// TIA Portal project "programa_plc_hmi_V16" (V16)

(* hardware
DEVICE "S71500/ET200MP station_1"  S7-1500 station
   slot 0: "Rail_0"  Rack  6ES7 590-1***0-0AA0
   slot 1: "PLC_1"  CPU 1513-1 PN  6ES7 513-1AL02-0AB0  V2.6
      slot 3: "CPU display_1"  6ES7591-1AA00-0AA0
   slot 2: "DI 16x24VDC BA_1"  DI 16x24VDC BA  6ES7 521-1BH10-0AA0  V1.0
   slot 3: "DQ 16x24VDC/0.5A BA_1"  DQ 16x24VDC/0.5A BA  6ES7 522-1BH10-0AA0  V1.0
   slot 4: "AI 4xU/I/RTD/TC / AQ 2xU/I ST_1"  AI/AQ 4xU/I/RTD/TC / 2xU/I ST  6ES7 534-7QE00-0AB0  V1.0
DEVICE "HMI_1"  KTP400 Comfort
   slot 0: "HMI_1"  KTP400 Comfort  6AV2 124-2DC01-0AX0  16.0.0.0
   slot 1: "HMI_RT_1"  KTP400 Comfort  6AV2 124-2DC01-0AX0  16.0.0.0
   slot 5: "HMI_1.IE_CP_1"  PROFINET Interface  16.0.0.0
      slot 1: "Interfaz PROFINET_1"  PROFINET Interface
         slot 1: "Port_1"  Port
   slot 7: "HMI_1.MPI/DP_CP_1"  MPI/DP Interface  16.0.0.0
*)

// ===== PLC "PLC_1"  CPU 1513-1 PN =====

VAR_GLOBAL   // PLC tag table "Default tag table"
   "System_Byte" AT %MB1 : Byte;
   "FirstScan" AT %M1.0 : Bool;
   "DiagStatusUpdate" AT %M1.1 : Bool;
   "AlwaysTRUE" AT %M1.2 : Bool;
   "AlwaysFALSE" AT %M1.3 : Bool;
   "Clock_Byte" AT %MB0 : Byte;
   "Clock_10Hz" AT %M0.0 : Bool;
   "Clock_5Hz" AT %M0.1 : Bool;
   "Clock_2.5Hz" AT %M0.2 : Bool;
   "Clock_2Hz" AT %M0.3 : Bool;
   "Clock_1.25Hz" AT %M0.4 : Bool;
   "Clock_1Hz" AT %M0.5 : Bool;
   "Clock_0.625Hz" AT %M0.6 : Bool;
   "Clock_0.5Hz" AT %M0.7 : Bool;
   "hmi star" AT %M200.0 : Bool;
   "hm1 led" AT %M200.1 : Bool;
END_VAR

VAR_GLOBAL   // PLC tag table "Conveyor_1"
   "c1_paro_de_emergencia" AT %I0.0 : Bool;
   "c1_barrera_de_seguridad" AT %I0.1 : Bool;
   "c1_variador_en_run" AT %I0.2 : Bool;
   "c1_auxiliar_guardamotor" AT %I0.3 : Bool;
   "c1_auxiliar_seccionador" AT %I0.4 : Bool;
   "c1_variador_en_falla" AT %I0.5 : Bool;
   "c1_pulsador_arranque" AT %I0.6 : Bool;
   "c1_pulsador_parada" AT %I0.7 : Bool;
   "c1_reset" AT %I1.0 : Bool;
   "c1_modo_auto_manual" AT %I1.1 : Bool;
   "c1_variador_a_run" AT %Q0.0 : Bool;
   "c1_sistema_en_automatico" AT %Q0.1 : Bool;
   "c1_sistema_en_manual" AT %Q0.2 : Bool;
   "c1_sistema_en_falla" AT %Q0.3 : Bool;
   "c1_sirena" AT %Q0.4 : Bool;
   "c1_reset_sistema" AT %Q0.5 : Bool;
   "c1_referencia_de_velocidad" AT %IW2 : Int;
   "c1_referencia_actual_velocidad" AT %QW2 : Int;
   "c1_falla_en_arraque" AT %M110.0 : Bool;
   "c1_auxiliar_conveyor_run" AT %M110.1 : Bool;
   "c1_indicador_conveyor_run" AT %Q0.6 : Bool;
   "c1_auxiliar_modo_automatico" AT %M110.3 : Bool;
   "c1_auxiliar_modo_manual" AT %M110.4 : Bool;
   "c1_auxiliar_start_manual" AT %M110.5 : Bool;
   "c1_auxiliar_start_auto" AT %M110.6 : Bool;
   "c1_paro_de_emergencia_m" AT %M100.0 : Bool;
   "c1_barrera_de_seguridad_m" AT %M100.1 : Bool;
   "c1_variador_en_run_m" AT %M100.2 : Bool;
   "c1_auxiliar_guardamotor_m" AT %M100.3 : Bool;
   "c1_auxiliar_seccionador_m" AT %M100.4 : Bool;
   "c1_variador_en_falla_m" AT %M100.5 : Bool;
   "c1_pulsador_arranque_m" AT %M100.6 : Bool;
   "c1_pulsador_parada_m" AT %M100.7 : Bool;
   "c1_reset_m" AT %M101.0 : Bool;
   "c1_modo_auto_manual_m" AT %M101.1 : Bool;
   "c1_variador_a_run_m" AT %M105.0 : Bool;
   "c1_sistema_en_automatico_m" AT %M105.1 : Bool;
   "c1_sistema_en_manual_m" AT %M105.2 : Bool;
   "c1_sistema_en_falla_m" AT %M105.3 : Bool;
   "c1_sirena_m" AT %M105.4 : Bool;
   "c1_reset_sistema_m" AT %M105.5 : Bool;
   "c1_indicador_conveyor_run_m" AT %M105.6 : Bool;
   "c1_referencia_de_velocidad_m" AT %MW150 : Word;
   "c1_referencia_actual_velocidad_m" AT %MW170 : Word;
   "c1_percentage input" AT %MW160 : Word;
   "c1_brazo_en_funcionamiento" AT %I1.2 : Bool;
   "c1_brazo_en_falla" AT %I1.3 : Bool;
   "c1_cnc_funcionamiento" AT %I1.4 : Bool;
   "c1_brazo_en_funcionamiento_m" AT %M101.2 : Bool;
   "c1_brazo_en_falla_m" AT %M101.3 : Bool;
   "c1_cnc_funcionamiento_m" AT %M101.4 : Bool;
   "c1_selector_producto" AT %Q0.7 : Bool;
   "c1_selector_producto_m" AT %M105.7 : Bool;
   "c1_sistema_cnc_1_en _funcinamiento" AT %M110.7 : Bool;
   "c1_sistema_cnc_1_en_falla" AT %M111.0 : Bool;
   "c1_sensor_producto_acabado" AT %I1.5 : Bool;
   "c1_sensor_producto_acabado_m" AT %M101.5 : Bool;
   "c1_cnc_arranque" AT %Q1.0 : Bool;
   "c1_cnc_parada" AT %Q1.1 : Bool;
   "c1_cnc_reset" AT %Q1.2 : Bool;
   "c1_cnc_arranque_m" AT %M106.0 : Bool;
   "c1_cnc_parada_m" AT %M106.1 : Bool;
   "c1_cnc_reset_m" AT %M106.2 : Bool;
   "c1_sensor_producto_entrada" AT %I1.6 : Bool;
   "c1_sensor_producto_entrada_m" AT %M101.6 : Bool;
   "c1_habilitar_material" AT %Q1.3 : Bool;
   "c1_habilitar_material_m" AT %M106.3 : Bool;
   "c1hmistart" AT %M210.0 : Bool;
   "c1hmiled" AT %M210.1 : Bool;
END_VAR

DATA_BLOCK "Direct_start_conveyor_1"   // DB1
{ S7_Optimized_Access := 'TRUE' }
VERSION : 0.1
// stored: InstanceOfName Direct_start
"Direct_start"
BEGIN
END_DATA_BLOCK

DATA_BLOCK "Percentage scaling_input_conveyor_1"   // DB2
{ S7_Optimized_Access := 'TRUE' }
VERSION : 0.1
// stored: InstanceOfName Percentage scaling
"Percentage scaling"
BEGIN
END_DATA_BLOCK

DATA_BLOCK "Cnc_operation_conveyor_1"   // DB4
{ S7_Optimized_Access := 'TRUE' }
VERSION : 0.1
// stored: InstanceOfName Cnc_operation
"Cnc_operation"
BEGIN
END_DATA_BLOCK

FUNCTION_BLOCK "Direct_start"   // FB1, LAD
{ S7_Optimized_Access := 'TRUE' }
VERSION : 0.1
   VAR_INPUT
      start : Bool;
      aux_emergency : Bool;
      aux_overload : Bool;
      aux_feedback : Bool;
      reset : Bool;
   END_VAR
   VAR_OUTPUT
      contactor_output : Bool;
      contactor_failure : Bool;
   END_VAR
   VAR
      aux_failure : Bool;
      aux_feedback_time_is_up : Bool;
      time_feedback : TON_TIME;
      motor_run : Bool;
   END_VAR
BEGIN

REGION Network 1
   // system failure
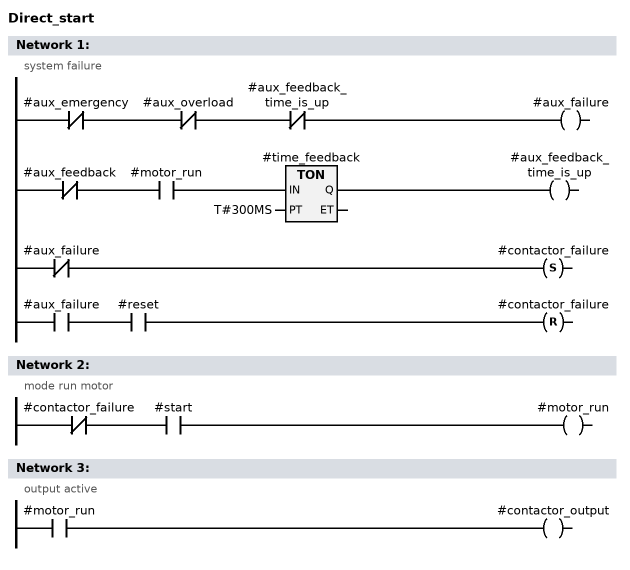
   #aux_failure := NOT #aux_emergency AND NOT #aux_overload AND NOT #aux_feedback_time_is_up;
   #time_feedback(IN := NOT #aux_feedback AND #motor_run, PT := T#300MS);   // TON
   #aux_feedback_time_is_up := #time_feedback.Q;
   IF NOT #aux_failure THEN #contactor_failure := TRUE; END_IF;
   IF #aux_failure AND #reset THEN #contactor_failure := FALSE; END_IF;
END_REGION

REGION Network 2
   // mode run motor
   RUNG wire#powerrail
      I_Contact( #contactor_failure )
      Contact( #start )
      Coil( #motor_run )
   END_RUNG
   // the same network as SCL:
   #motor_run := NOT #contactor_failure AND #start;
END_REGION

REGION Network 3
   // output active
   RUNG wire#powerrail
      Contact( #motor_run )
      Coil( #contactor_output )
   END_RUNG
   // the same network as SCL:
   #contactor_output := #motor_run;
END_REGION
END_FUNCTION_BLOCK

FUNCTION_BLOCK "Percentage scaling"   // FB2, LAD
{ S7_Optimized_Access := 'TRUE' }
VERSION : 0.1
   VAR_INPUT
      analog_sign : Word;
   END_VAR
   VAR_OUTPUT
      escalated_signal : Int;
   END_VAR
   VAR
      norm_scale : Real;
   END_VAR
BEGIN

REGION Network 1
   // scale the analog signal pulses to a percentage from 0 to 100%
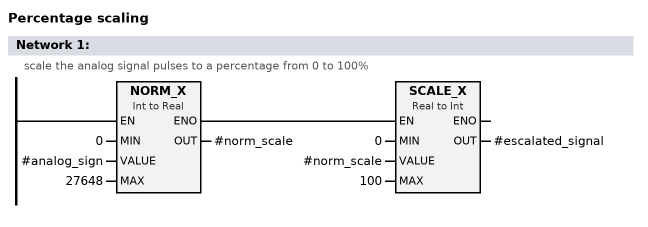
   RUNG wire#powerrail
      { S7_Templates := "[SrcType := Int, DestType := Real]" } Normalize(min := 0, value := #analog_sign, max := 27648, out => #norm_scale)
      { S7_Templates := "[SrcType := Real, DestType := Int]" } Scale(min := 0, value := #norm_scale, max := 100, out => #escalated_signal)
   END_RUNG
   // the same network as SCL:
   #norm_scale := NORM_X(MIN := 0, VALUE := #analog_sign, MAX := 27648);
   #escalated_signal := SCALE_X(MIN := 0, VALUE := #norm_scale, MAX := 100);
END_REGION
END_FUNCTION_BLOCK

FUNCTION_BLOCK "Cnc_operation"   // FB3, LAD
{ S7_Optimized_Access := 'TRUE' }
VERSION : 0.1
// start -up operation
   VAR_INPUT
      start : Bool;
      stop : Bool;
      reset : Bool;
      feedbacks_operation : Bool;
      fault : Bool;
      sensor_output : Bool;
      sensor_input : Bool;
      cnc_operation : Bool;
   END_VAR
   VAR_OUTPUT
      system_cnc_run : Bool;
      system_cnc_stop : Bool;
      system_cnc_reset : Bool;
      system_cnc_operation : Bool;
      system_cnc_fault : Bool;
   END_VAR
   VAR
      start_operation : Bool;
      set_fault : Bool;
      stop_operation : Bool;
      aux_stop_operation : Bool;
      operation_restart_time : TON_TIME;
      aux_reset : Bool;
      aux_sensor_input : Bool;
      aux_sensor_output : Bool;
      time_sensor_input : TON_TIME;
   END_VAR
BEGIN

REGION Network 1
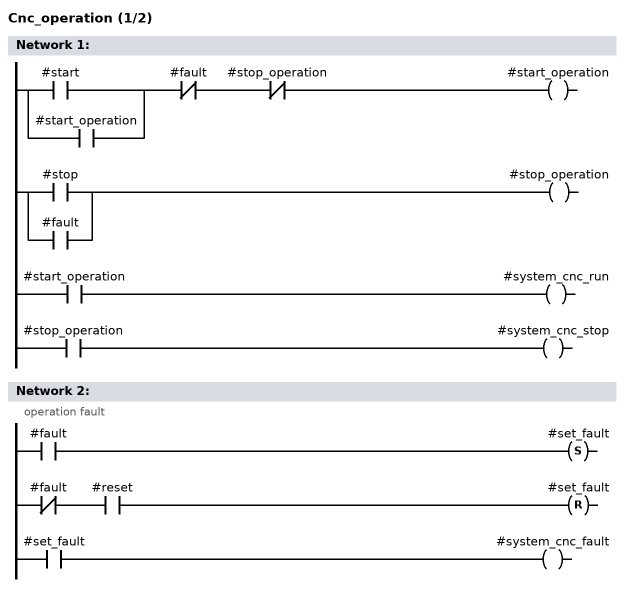
   RUNG wire#powerrail
      Contact( #start )
      wire#w1
      I_Contact( #fault )
      I_Contact( #stop_operation )
      Coil( #start_operation )
   END_RUNG
   RUNG wire#powerrail
      Contact( #start_operation )
   END_RUNG wire#w1
   RUNG wire#powerrail
      Contact( #stop )
      wire#w2
      Coil( #stop_operation )
   END_RUNG
   RUNG wire#powerrail
      Contact( #fault )
   END_RUNG wire#w2
   RUNG wire#powerrail
      Contact( #start_operation )
      Coil( #system_cnc_run )
   END_RUNG
   RUNG wire#powerrail
      Contact( #stop_operation )
      Coil( #system_cnc_stop )
   END_RUNG
   // the same network as SCL:
   #start_operation := (#start OR #start_operation) AND NOT #fault AND NOT #stop_operation;
   #stop_operation := #stop OR #fault;
   #system_cnc_run := #start_operation;
   #system_cnc_stop := #stop_operation;
END_REGION

REGION Network 2
   // operation fault
   RUNG wire#powerrail
      Contact( #fault )
      S_Coil( #set_fault )
   END_RUNG
   RUNG wire#powerrail
      I_Contact( #fault )
      Contact( #reset )
      R_Coil( #set_fault )
   END_RUNG
   RUNG wire#powerrail
      Contact( #set_fault )
      Coil( #system_cnc_fault )
   END_RUNG
   // the same network as SCL:
   IF #fault THEN #set_fault := TRUE; END_IF;
   IF NOT #fault AND #reset THEN #set_fault := FALSE; END_IF;
   #system_cnc_fault := #set_fault;
END_REGION

REGION Network 3
   // feedbacks operation
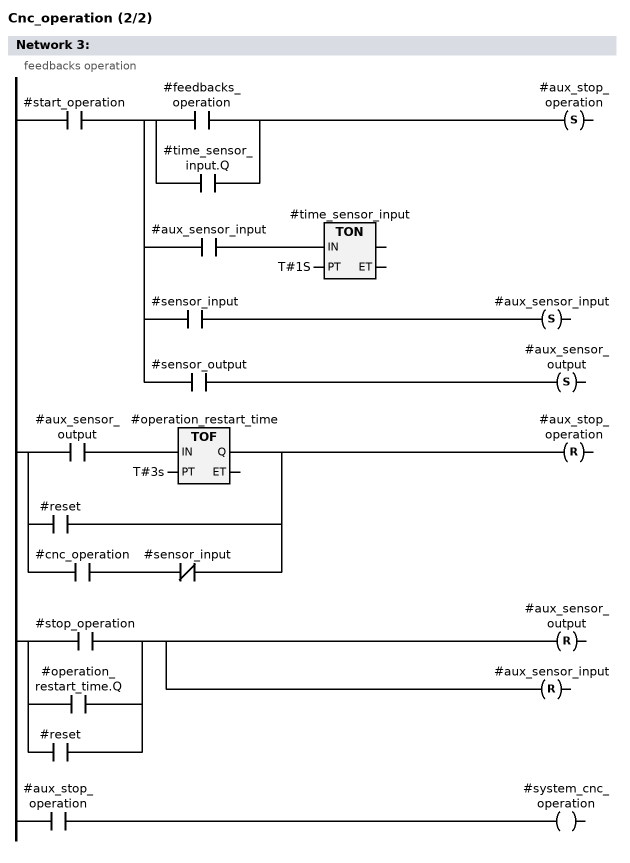
   IF #start_operation AND (#feedbacks_operation OR #time_sensor_input.Q) THEN
       #aux_stop_operation := TRUE;
   END_IF;
   #time_sensor_input(IN := #start_operation AND #aux_sensor_input, PT := T#1S);   // TON
   IF #start_operation AND #sensor_input THEN #aux_sensor_input := TRUE; END_IF;
   IF #start_operation AND #sensor_output THEN #aux_sensor_output := TRUE; END_IF;
   #operation_restart_time(IN := #aux_sensor_output, PT := T#3s);   // TOF
   IF #operation_restart_time.Q OR #reset OR (#cnc_operation AND NOT #sensor_input) THEN
       #aux_stop_operation := FALSE;
   END_IF;
   IF #stop_operation OR #operation_restart_time.Q OR #reset THEN
       #aux_sensor_output := FALSE;
       #aux_sensor_input := FALSE;
   END_IF;
   #system_cnc_operation := #aux_stop_operation;
END_REGION
END_FUNCTION_BLOCK

FUNCTION "Conveyor_1" : Void   // FC1, LAD
{ S7_Optimized_Access := 'TRUE' }
VERSION : 0.1
BEGIN

REGION Network 1
   // Start motor conveyor 1
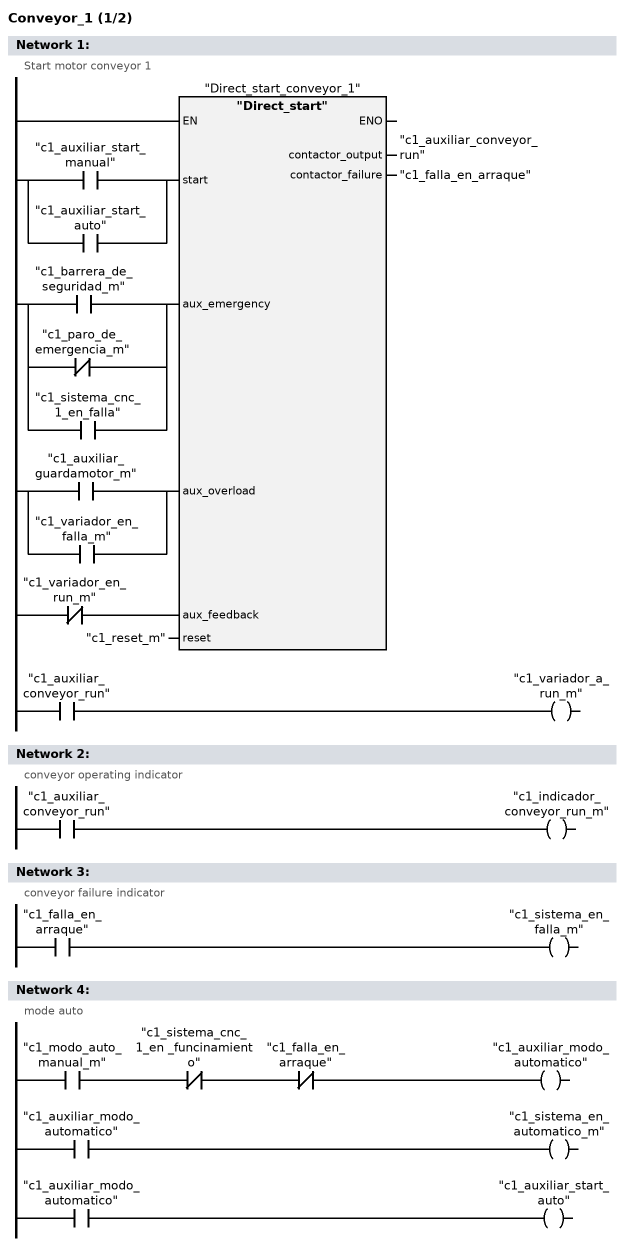
   RUNG wire#powerrail
      "Direct_start_conveyor_1"(start := wire#w1, aux_emergency := wire#w2, aux_overload := wire#w3, aux_feedback := wire#w4, reset := "c1_reset_m", contactor_output => "c1_auxiliar_conveyor_run", contactor_failure => "c1_falla_en_arraque")
   END_RUNG
   RUNG wire#powerrail
      Contact( "c1_auxiliar_start_manual" )
   END_RUNG wire#w1
   RUNG wire#powerrail
      Contact( "c1_auxiliar_start_auto" )
   END_RUNG wire#w1
   RUNG wire#powerrail
      Contact( "c1_barrera_de_seguridad_m" )
   END_RUNG wire#w2
   RUNG wire#powerrail
      I_Contact( "c1_paro_de_emergencia_m" )
   END_RUNG wire#w2
   RUNG wire#powerrail
      Contact( "c1_sistema_cnc_1_en_falla" )
   END_RUNG wire#w2
   RUNG wire#powerrail
      Contact( "c1_auxiliar_guardamotor_m" )
   END_RUNG wire#w3
   RUNG wire#powerrail
      Contact( "c1_variador_en_falla_m" )
   END_RUNG wire#w3
   RUNG wire#powerrail
      I_Contact( "c1_variador_en_run_m" )
   END_RUNG wire#w4
   RUNG wire#powerrail
      Contact( "c1_auxiliar_conveyor_run" )
      Coil( "c1_variador_a_run_m" )
   END_RUNG
   // the same network as SCL:
   "Direct_start_conveyor_1"(start := "c1_auxiliar_start_manual" OR "c1_auxiliar_start_auto",   // "Direct_start"
                           aux_emergency := "c1_barrera_de_seguridad_m" OR NOT "c1_paro_de_emergencia_m" OR "c1_sistema_cnc_1_en_falla",
                           aux_overload := "c1_auxiliar_guardamotor_m" OR "c1_variador_en_falla_m",
                           aux_feedback := NOT "c1_variador_en_run_m",
                           reset := "c1_reset_m",
                           contactor_output => "c1_auxiliar_conveyor_run",
                           contactor_failure => "c1_falla_en_arraque");
   "c1_variador_a_run_m" := "c1_auxiliar_conveyor_run";
END_REGION

REGION Network 2
   // conveyor operating indicator
   RUNG wire#powerrail
      Contact( "c1_auxiliar_conveyor_run" )
      Coil( "c1_indicador_conveyor_run_m" )
   END_RUNG
   // the same network as SCL:
   "c1_indicador_conveyor_run_m" := "c1_auxiliar_conveyor_run";
END_REGION

REGION Network 3
   // conveyor failure indicator
   RUNG wire#powerrail
      Contact( "c1_falla_en_arraque" )
      Coil( "c1_sistema_en_falla_m" )
   END_RUNG
   // the same network as SCL:
   "c1_sistema_en_falla_m" := "c1_falla_en_arraque";
END_REGION

REGION Network 4
   // mode auto
   RUNG wire#powerrail
      Contact( "c1_modo_auto_manual_m" )
      I_Contact( "c1_sistema_cnc_1_en _funcinamiento" )
      I_Contact( "c1_falla_en_arraque" )
      Coil( "c1_auxiliar_modo_automatico" )
   END_RUNG
   RUNG wire#powerrail
      Contact( "c1_auxiliar_modo_automatico" )
      Coil( "c1_sistema_en_automatico_m" )
   END_RUNG
   RUNG wire#powerrail
      Contact( "c1_auxiliar_modo_automatico" )
      Coil( "c1_auxiliar_start_auto" )
   END_RUNG
   // the same network as SCL:
   "c1_auxiliar_modo_automatico" := "c1_modo_auto_manual_m" AND NOT "c1_sistema_cnc_1_en _funcinamiento" AND NOT "c1_falla_en_arraque";
   "c1_sistema_en_automatico_m" := "c1_auxiliar_modo_automatico";
   "c1_auxiliar_start_auto" := "c1_auxiliar_modo_automatico";
END_REGION

REGION Network 5
   // system hand
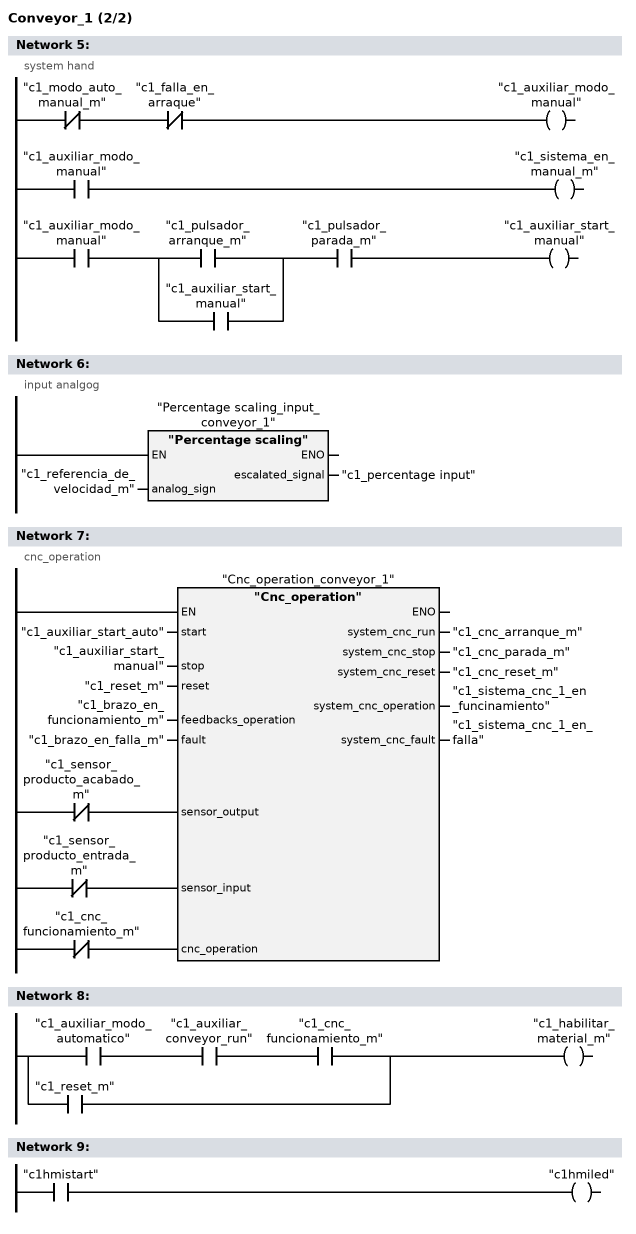
   RUNG wire#powerrail
      I_Contact( "c1_modo_auto_manual_m" )
      I_Contact( "c1_falla_en_arraque" )
      Coil( "c1_auxiliar_modo_manual" )
   END_RUNG
   RUNG wire#powerrail
      Contact( "c1_auxiliar_modo_manual" )
      Coil( "c1_sistema_en_manual_m" )
   END_RUNG
   RUNG wire#powerrail
      Contact( "c1_auxiliar_modo_manual" )
      wire#w1
      Contact( "c1_pulsador_arranque_m" )
      wire#w2
      Contact( "c1_pulsador_parada_m" )
      Coil( "c1_auxiliar_start_manual" )
   END_RUNG
   RUNG wire#w1
      Contact( "c1_auxiliar_start_manual" )
   END_RUNG wire#w2
   // the same network as SCL:
   "c1_auxiliar_modo_manual" := NOT "c1_modo_auto_manual_m" AND NOT "c1_falla_en_arraque";
   "c1_sistema_en_manual_m" := "c1_auxiliar_modo_manual";
   "c1_auxiliar_start_manual" := "c1_auxiliar_modo_manual" AND ("c1_pulsador_arranque_m" OR "c1_auxiliar_start_manual") AND "c1_pulsador_parada_m";
END_REGION

REGION Network 6
   // input analgog
   RUNG wire#powerrail
      "Percentage scaling_input_conveyor_1"(analog_sign := "c1_referencia_de_velocidad_m", escalated_signal => "c1_percentage input")
   END_RUNG
   // the same network as SCL:
   "Percentage scaling_input_conveyor_1"(analog_sign := "c1_referencia_de_velocidad_m",   // "Percentage scaling"
                           escalated_signal => "c1_percentage input");
END_REGION

REGION Network 7
   // cnc_operation
   RUNG wire#powerrail
      "Cnc_operation_conveyor_1"(sensor_output := wire#w1, sensor_input := wire#w2, cnc_operation := wire#w3, start := "c1_auxiliar_start_auto", stop := "c1_auxiliar_start_manual", reset := "c1_reset_m", feedbacks_operation := "c1_brazo_en_funcionamiento_m", fault := "c1_brazo_en_falla_m", system_cnc_run => "c1_cnc_arranque_m", system_cnc_stop => "c1_cnc_parada_m", system_cnc_reset => "c1_cnc_reset_m", system_cnc_operation => "c1_sistema_cnc_1_en _funcinamiento", system_cnc_fault => "c1_sistema_cnc_1_en_falla")
   END_RUNG
   RUNG wire#powerrail
      I_Contact( "c1_sensor_producto_acabado_m" )
   END_RUNG wire#w1
   RUNG wire#powerrail
      I_Contact( "c1_sensor_producto_entrada_m" )
   END_RUNG wire#w2
   RUNG wire#powerrail
      I_Contact( "c1_cnc_funcionamiento_m" )
   END_RUNG wire#w3
   // the same network as SCL:
   "Cnc_operation_conveyor_1"(start := "c1_auxiliar_start_auto",   // "Cnc_operation"
                           stop := "c1_auxiliar_start_manual",
                           reset := "c1_reset_m",
                           feedbacks_operation := "c1_brazo_en_funcionamiento_m",
                           fault := "c1_brazo_en_falla_m",
                           sensor_output := NOT "c1_sensor_producto_acabado_m",
                           sensor_input := NOT "c1_sensor_producto_entrada_m",
                           cnc_operation := NOT "c1_cnc_funcionamiento_m",
                           system_cnc_run => "c1_cnc_arranque_m",
                           system_cnc_stop => "c1_cnc_parada_m",
                           system_cnc_reset => "c1_cnc_reset_m",
                           system_cnc_operation => "c1_sistema_cnc_1_en _funcinamiento",
                           system_cnc_fault => "c1_sistema_cnc_1_en_falla");
END_REGION

REGION Network 8
   RUNG wire#powerrail
      Contact( "c1_auxiliar_modo_automatico" )
      Contact( "c1_auxiliar_conveyor_run" )
      Contact( "c1_cnc_funcionamiento_m" )
      wire#w1
      Coil( "c1_habilitar_material_m" )
   END_RUNG
   RUNG wire#powerrail
      Contact( "c1_reset_m" )
   END_RUNG wire#w1
   // the same network as SCL:
   "c1_habilitar_material_m" := ("c1_auxiliar_modo_automatico" AND "c1_auxiliar_conveyor_run" AND "c1_cnc_funcionamiento_m") OR "c1_reset_m";
END_REGION

REGION Network 9
   RUNG wire#powerrail
      Contact( "c1hmistart" )
      Coil( "c1hmiled" )
   END_RUNG
   // the same network as SCL:
   "c1hmiled" := "c1hmistart";
END_REGION
END_FUNCTION

ORGANIZATION_BLOCK "Main"   // OB1, LAD, ProgramCycle
TITLE = "Main Program Sweep (Cycle)"
{ S7_Optimized_Access := 'TRUE' }
VERSION : 0.1
   VAR_INPUT
      Initial_Call : Bool;   // Initial call of this OB
      Remanence : Bool;   // =True, if remanent data are available
   END_VAR
BEGIN

REGION Network 1
   // Conveyor line 1
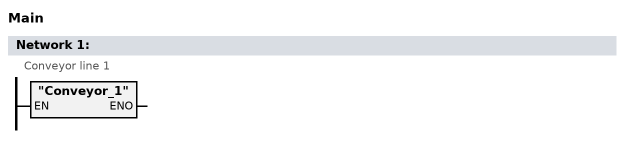
   RUNG wire#powerrail
      "Conveyor_1"()
   END_RUNG
   // the same network as SCL:
   "Conveyor_1"();
END_REGION
END_ORGANIZATION_BLOCK

ORGANIZATION_BLOCK "Input_digital_memory"   // OB123, STL, ProgramCycle
TITLE = "Main Program Sweep (Cycle)"
{ S7_Optimized_Access := 'TRUE' }
VERSION : 0.1
   VAR_INPUT
      Initial_Call : Bool;   // Initial call of this OB
      Remanence : Bool;   // =True, if remanent data are available
   END_VAR
BEGIN

REGION Network 1
         A     "c1_paro_de_emergencia";
         =     "c1_paro_de_emergencia_m";
         A     "c1_barrera_de_seguridad";
         =     "c1_barrera_de_seguridad_m";
         A     "c1_variador_en_run";
         =     "c1_variador_en_run_m";
         A     "c1_auxiliar_guardamotor";
         =     "c1_auxiliar_guardamotor_m";
         A     "c1_auxiliar_seccionador";
         =     "c1_auxiliar_seccionador_m";
         A     "c1_variador_en_falla";
         =     "c1_variador_en_falla_m";
         A     "c1_pulsador_arranque";
         =     "c1_pulsador_arranque_m";
         A     "c1_pulsador_parada";
         =     "c1_pulsador_parada_m";
         A     "c1_reset";
         =     "c1_reset_m";
         A     "c1_modo_auto_manual";
         =     "c1_modo_auto_manual_m";
         A     "c1_brazo_en_funcionamiento";
         =     "c1_brazo_en_funcionamiento_m";
         A     "c1_brazo_en_falla";
         =     "c1_brazo_en_falla_m";
         A     "c1_cnc_funcionamiento";
         =     "c1_cnc_funcionamiento_m";
         A     "c1_sensor_producto_acabado";
         =     "c1_sensor_producto_acabado_m";
         A     "c1_sensor_producto_entrada";
         =     "c1_sensor_producto_entrada_m";
END_REGION
END_ORGANIZATION_BLOCK

ORGANIZATION_BLOCK "Input_analog_memory"   // OB124, STL, ProgramCycle
TITLE = "Main Program Sweep (Cycle)"
{ S7_Optimized_Access := 'TRUE' }
VERSION : 0.1
   VAR_INPUT
      Initial_Call : Bool;   // Initial call of this OB
      Remanence : Bool;   // =True, if remanent data are available
   END_VAR
BEGIN

REGION Network 1
         L     "c1_referencia_de_velocidad";
         T     "c1_referencia_actual_velocidad_m";
END_REGION
END_ORGANIZATION_BLOCK

ORGANIZATION_BLOCK "Output_digital_memory"   // OB125, STL, ProgramCycle
TITLE = "Main Program Sweep (Cycle)"
{ S7_Optimized_Access := 'TRUE' }
VERSION : 0.1
   VAR_INPUT
      Initial_Call : Bool;   // Initial call of this OB
      Remanence : Bool;   // =True, if remanent data are available
   END_VAR
BEGIN

REGION Network 1
         A     "c1_variador_a_run_m";
         =     "c1_variador_a_run";
         A     "c1_sistema_en_automatico_m";
         =     "c1_sistema_en_automatico";
         A     "c1_sistema_en_manual_m";
         =     "c1_sistema_en_manual";
         A     "c1_sistema_en_falla_m";
         =     "c1_sistema_en_falla";
         A     "c1_sirena_m";
         =     "c1_sirena";
         A     "c1_reset_sistema_m";
         =     "c1_reset_sistema";
         A     "c1_indicador_conveyor_run_m";
         =     "c1_indicador_conveyor_run";
         A     "c1_selector_producto_m";
         =     "c1_selector_producto";
         A     "c1_cnc_arranque_m";
         =     "c1_cnc_arranque";
         A     "c1_cnc_parada_m";
         =     "c1_cnc_parada";
         A     "c1_cnc_reset_m";
         =     "c1_cnc_reset";
         A     "c1_habilitar_material_m";
         =     "c1_habilitar_material";
END_REGION
END_ORGANIZATION_BLOCK

ORGANIZATION_BLOCK "Output_analog_memory"   // OB126, STL, ProgramCycle
TITLE = "Main Program Sweep (Cycle)"
{ S7_Optimized_Access := 'TRUE' }
VERSION : 0.1
   VAR_INPUT
      Initial_Call : Bool;   // Initial call of this OB
      Remanence : Bool;   // =True, if remanent data are available
   END_VAR
BEGIN

REGION Network 1
         L     "c1_referencia_de_velocidad_m";
         T     "c1_referencia_actual_velocidad";
END_REGION
END_ORGANIZATION_BLOCK

(* ===== HMI "HMI_RT_1" =====
system functions are stored by id; their names below are inferred from use
connection "HMI_Conexión_1": ETHERNET, S7_1500_OMS

HMI tags "Tabla de variables estándar"
   "c1hmistart" : Bool = PLC c1hmistart AT %M210.0, 1 s
   "c1hmiled" : Bool = PLC c1hmiled AT %M210.1, 1 s

screen "Imagen raíz" 480x212, template "Plantilla_1"
   on GenerateScreen: SetTag("Número_imagen_variable", 1)
   Button "Botón_1" at 28,28 size 96x32; TextOff 'on'
      on Press: SetBit("c1hmistart")
   Circle "Círculo_1" at 202,36 size 48x48
      Appearance <- "c1hmiled"

Template "Plantilla_1" 480x212
   Button "Exit" at 379,148 size 63x63; TextOff 'Exit'; PictureOff "ExitRuntime_KTP400_Comfort_TR"; PictureOn "ExitRuntime_KTP400_Comfort_TR"
      on Release: StopRuntime(0)
   Button "Log on" at 265,148 size 63x63; TextOff 'Log on'; PictureOff "Login_KTP400_Comfort_TR"; PictureOn "Login_KTP400_Comfort_TR"
      on Release: function_a2a04561()
   Button "Language" at 151,148 size 63x63; TextOff 'Language'; PictureOff "ToggleLanguage_KTP400_Comfort_TR"; PictureOn "ToggleLanguage_KTP400_Comfort_TR"
      on Release: function_fb9197e8(-1)
   Button "Start screen" at 37,148 size 63x63; TextOff 'Start screen'; PictureOff "NavigateHome_KTP400_Comfort_TR"; PictureOn "NavigateHome_KTP400_Comfort_TR"
      on Release: ActivateScreen("Imagen raíz", 0)
*)